(* CODESYS project io.library
   Company: Red&Blue Company
   DefaultNamespace: IO
   Version: 0.1.0.0
   Placeholder: Inputs and outputs
   Author: LeHoaiVuong
   Description: This library holds functionality for sensors and actuators,
   Title: Inputs and outputs

Project tree, tasks and I/O mapping:
  libraries: Tc2_Standard, * (Beckhoff Automation GmbH); Tc2_System, * (Beckhoff Automation GmbH); Tc3_Module, * (Beckhoff Automation GmbH)
  DUTs/
  GVLs/
  POUs/
    function block FB_O5D100 [ST]
  Version/
    global variables Global_Version
*)

// Version/Global_Version
{attribute 'TcGenerated'}
{attribute 'no-analysis'}
{attribute 'linkalways'}
// This function has been automatically generated from the project information.
VAR_GLOBAL CONSTANT
	{attribute 'const_non_replaced'}
	stLibVersion_Inputs_and_outputs : ST_LibVersion := (iMajor := 0, iMinor := 1, iBuild := 0, iRevision := 0, nFlags := 0, sVersion := '0.1.0.0');
END_VAR

// POUs/FB_O5D100
FUNCTION_BLOCK FB_O5D100
VAR_OUTPUT
	nDistance : INT; //[cm]
	nInSwitchPoint : BOOL; //[True if below 100cm]
END_VAR
VAR
	aInputBytes AT %I* : ARRAY[1..2] OF BYTE;
	nWord1 : WORD;
	nWord2 : WORD;
	nWord3 : WORD;
END_VAR

nWord1 := TO_WORD(aInputBytes[1]);


nWord2 := TO_WORD(aInputBytes[2]);
nInSwitchPoint := aInputBytes[2].0;

nWord1 := SHL(nWord1, 8);

nWord3 := nWord1 OR nWord2;

nWord3 := SHL(nWord3, 4);

nDistance := TO_INT(nWord3);

END_FUNCTION_BLOCK
